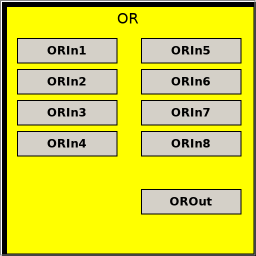
VISUALIZATION V_PH_OR  // 256x256
VAR_INPUT
	stSafetyOR			:ST_SAFETY_FBOR;
	
END_VAR
    Rectangle (2,2 256x256), colour toggle: stSafetyOR.bGeneralError
    Label (5,6 246x25), "OR"
    RoundedRectangle (17,38 100x25), "ORIn1", colour toggle: stSafetyOR.uStatus.stStatusWords.wInputs.8
    RoundedRectangle (17,100 100x25), "ORIn3", colour toggle: stSafetyOR.uStatus.stStatusWords.wInputs.10
    RoundedRectangle (17,131 100x25), "ORIn4", colour toggle: stSafetyOR.uStatus.stStatusWords.wInputs.11
    RoundedRectangle (141,38 100x25), "ORIn5", colour toggle: stSafetyOR.uStatus.stStatusWords.wInputs.12
    RoundedRectangle (141,69 100x25), "ORIn6", colour toggle: stSafetyOR.uStatus.stStatusWords.wInputs.13
    RoundedRectangle (141,100 100x25), "ORIn7", colour toggle: stSafetyOR.uStatus.stStatusWords.wInputs.14
    RoundedRectangle (141,131 100x25), "ORIn8", colour toggle: stSafetyOR.uStatus.stStatusWords.wInputs.15
    RoundedRectangle (17,69 100x25), "ORIn2", colour toggle: stSafetyOR.uStatus.stStatusWords.wInputs.9
    RoundedRectangle (141,189 100x25), "OROut", colour toggle: stSafetyOR.uStatus.stStatusWords.wOutputs.0
    Textfield (17,226 234x25), text list: 'TL_FbState', text index: stSafetyOR.eState
END_VISUALIZATION

(* stored: Version 1.1.0.1, ProductVersion 3.1.4024.4
   Visu V_PH_OR: Id {1473c0c0-8d71-44c9-9b18-a749729e6038} *)
